ABB RobotStudio station: Assingmennt.rspag

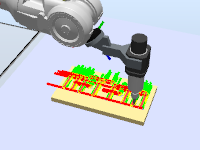
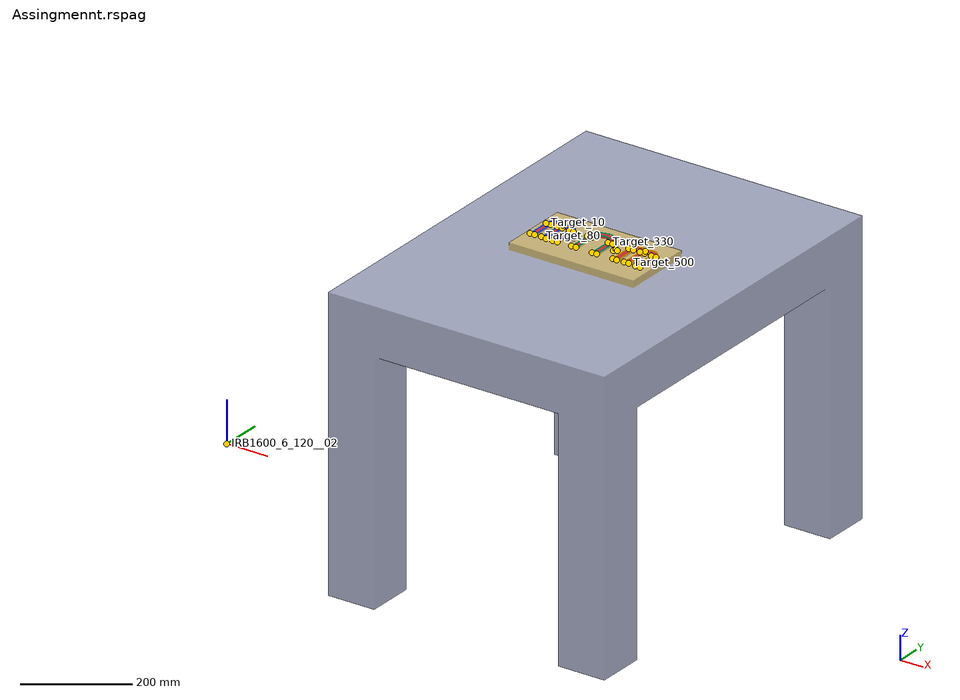
[picture v1: parts stored in the station drawn from their meshes, with robot base, taught points and paths (robot models come from the ABB library and are not in the file)]
--- station ---
Station Assingmennt (saved by RobotStudio 22.1.9826.0)
Controller IRB1600_6_120
  mechanical unit ROB_1: IRB1600_6_120__02, 6 joints, base frame (0, 0, 0) mm
Layout (positions relative to the parent item):
  - IRB1600_6_120__02 [mechanism, from Robots\IRB1600_6_120_G_02.rslib] at (0, 0, 0) mm; joint values [-0.0435, -0.0082, 0.1583, 0.0389, 0.7583, -0.0625] (rad or m)
  - MyTool [mechanism, from Training Objects\myTool.rslib] at (778.67, -32.12, 820.53) mm, rotated rx 180 ry 38 rz 180 deg
  - Table [part] at (800, 0, 0) mm, rotated rx 0 ry 0 rz 90 deg, size 800 x 600 x 600 mm
  - Part1 [part] at (800, 0, 600) mm, size 270 x 150 x 20 mm
Attachment: MyTool is attached to IRB1600_6_120__02 / Link6
Targets, tools, work objects and paths stored in the station and not in the controller backup, written as RAPID:
! task T_ROB1
MODULE Module1
  CONST robtarget Target_60:=[[202.210676312,424.371338975,20],[0,0,1,0],[0,0,0,0],[9E+09,9E+09,9E+09,9E+09,9E+09,9E+09]];
  CONST robtarget Target_120:=[[227.210676312,424.371338975,20],[0,0,1,0],[0,0,0,0],[9E+09,9E+09,9E+09,9E+09,9E+09,9E+09]];
  CONST robtarget Target_180:=[[222.399357136,434.659053801,20],[0,0,1,0],[0,0,0,0],[9E+09,9E+09,9E+09,9E+09,9E+09,9E+09]];
  CONST robtarget Target_210:=[[186.309791958,430.022914141,20],[0,0,1,0],[0,0,0,0],[9E+09,9E+09,9E+09,9E+09,9E+09,9E+09]];
  CONST robtarget Target_320:=[[307.210676312,433.031593012,20],[0,0,1,0],[0,0,0,0],[9E+09,9E+09,9E+09,9E+09,9E+09,9E+09]];
  CONST robtarget Target_380:=[[284.710676312,441.69184705,20],[0,0,1,0],[0,0,0,0],[9E+09,9E+09,9E+09,9E+09,9E+09,9E+09]];
  CONST robtarget Target_530:=[[406.25,424.371338975,20],[0,0,1,0],[0,0,0,0],[9E+09,9E+09,9E+09,9E+09,9E+09,9E+09]];
  CONST robtarget Target_590:=[[401.499668485,434.138320297,20],[0,0,1,0],[0,0,0,0],[9E+09,9E+09,9E+09,9E+09,9E+09,9E+09]];
  CONST robtarget Target_620:=[[365.571673376,430.19199697,20],[0,0,1,0],[0,0,0,0],[9E+09,9E+09,9E+09,9E+09,9E+09,9E+09]];
  CONST robtarget Target_680:=[[381.25,424.371338975,20],[0,0,1,0],[0,0,0,0],[9E+09,9E+09,9E+09,9E+09,9E+09,9E+09]];
ENDMODULE


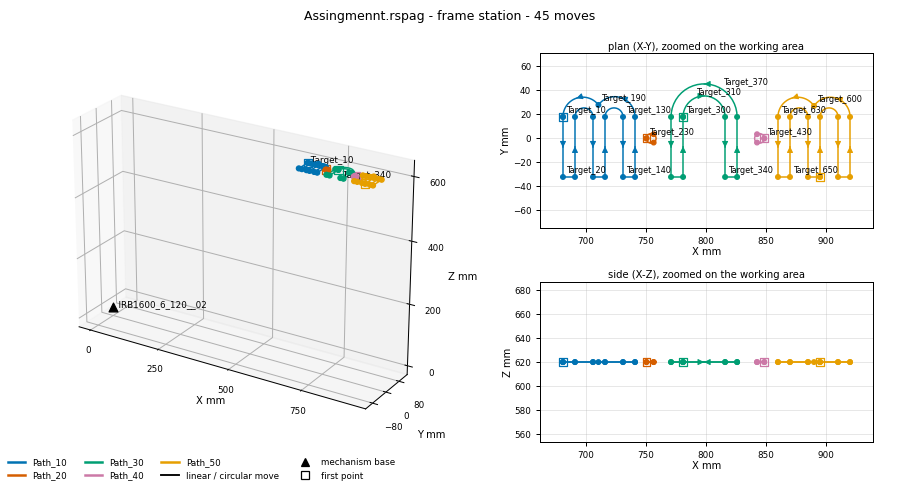
[picture p0: tool path of Assingmennt.rspag in frame station, 45 of 45 moves have a stored position in this frame; points joined in program order, loops and branches not executed]
--- Backups/IRB1600_6_120/RAPID/TASK1/PROGMOD/CalibData.mod ---
MODULE CalibData
    PERS tooldata MyTool:=[TRUE,[[31.792631019,0,229.638935148],[0.945518576,0,0.325568154,0]],[1,[0,0,1],[1,0,0,0],0,0,0]];
    PERS wobjdata Workobject_1:=[FALSE,TRUE,"",[[500,-400,600],[1,0,0,0]],[[0,0,0],[1,0,0,0]]];
ENDMODULE

--- Backups/IRB1600_6_120/RAPID/TASK1/PROGMOD/Module1.mod ---
MODULE Module1
    CONST robtarget Target_10:=[[180.960676312,417.876148446,20],[0,0,1,0],[0,0,0,0],[9E+09,9E+09,9E+09,9E+09,9E+09,9E+09]];
    CONST robtarget Target_20:=[[180.960676312,367.876148446,20],[0,0,1,0],[0,0,0,0],[9E+09,9E+09,9E+09,9E+09,9E+09,9E+09]];
    CONST robtarget Target_30:=[[190.960676312,367.876148446,20],[0,0,1,0],[0,0,0,0],[9E+09,9E+09,9E+09,9E+09,9E+09,9E+09]];
    CONST robtarget Target_40:=[[190.960676312,417.876148446,20],[0,0,1,0],[0,0,0,0],[9E+09,9E+09,9E+09,9E+09,9E+09,9E+09]];
    CONST robtarget Target_50:=[[194.710676312,424.371338975,20],[0,0,1,0],[0,0,0,0],[9E+09,9E+09,9E+09,9E+09,9E+09,9E+09]];
    CONST robtarget Target_70:=[[205.960676312,417.876148446,20],[0,0,1,0],[0,0,0,0],[9E+09,9E+09,9E+09,9E+09,9E+09,9E+09]];
    CONST robtarget Target_80:=[[205.960676312,367.876148446,20],[0,0,1,0],[0,0,0,0],[9E+09,9E+09,9E+09,9E+09,9E+09,9E+09]];
    CONST robtarget Target_90:=[[215.960676312,367.876148446,20],[0,0,1,0],[0,0,0,0],[9E+09,9E+09,9E+09,9E+09,9E+09,9E+09]];
    CONST robtarget Target_100:=[[215.960676312,417.876148446,20],[0,0,1,0],[0,0,0,0],[9E+09,9E+09,9E+09,9E+09,9E+09,9E+09]];
    CONST robtarget Target_110:=[[219.710676312,424.371338975,20],[0,0,1,0],[0,0,0,0],[9E+09,9E+09,9E+09,9E+09,9E+09,9E+09]];
    CONST robtarget Target_130:=[[230.960676312,417.876148446,20],[0,0,1,0],[0,0,0,0],[9E+09,9E+09,9E+09,9E+09,9E+09,9E+09]];
    CONST robtarget Target_140:=[[230.960676312,367.876148446,20],[0,0,1,0],[0,0,0,0],[9E+09,9E+09,9E+09,9E+09,9E+09,9E+09]];
    CONST robtarget Target_150:=[[240.960676312,367.876148446,20],[0,0,1,0],[0,0,0,0],[9E+09,9E+09,9E+09,9E+09,9E+09,9E+09]];
    CONST robtarget Target_160:=[[240.960676312,417.876148446,20],[0,0,1,0],[0,0,0,0],[9E+09,9E+09,9E+09,9E+09,9E+09,9E+09]];
    CONST robtarget Target_170:=[[235.405653207,430.388027618,20],[0,0,1,0],[0,0,0,0],[9E+09,9E+09,9E+09,9E+09,9E+09,9E+09]];
    CONST robtarget Target_190:=[[210.508284978,427.876148446,20],[0,0,1,0],[0,0,0,0],[9E+09,9E+09,9E+09,9E+09,9E+09,9E+09]];
    CONST robtarget Target_200:=[[198.881728,434.277720743,20],[0,0,1,0],[0,0,0,0],[9E+09,9E+09,9E+09,9E+09,9E+09,9E+09]];
    CONST robtarget Target_220:=[[180.960676312,417.876148446,20],[0,0,1,0],[0,0,0,0],[9E+09,9E+09,9E+09,9E+09,9E+09,9E+09]];
    CONST robtarget Target_230:=[[250.482336293,400,20],[0,0,1,0],[0,0,0,0],[9E+09,9E+09,9E+09,9E+09,9E+09,9E+09]];
    CONST robtarget Target_240:=[[252.482336293,403.464101615,20],[0,0,1,0],[0,0,0,0],[9E+09,9E+09,9E+09,9E+09,9E+09,9E+09]];
    CONST robtarget Target_250:=[[256.482336293,403.464101615,20],[0,0,1,0],[0,0,0,0],[9E+09,9E+09,9E+09,9E+09,9E+09,9E+09]];
    CONST robtarget Target_260:=[[258.482336293,400,20],[0,0,1,0],[0,0,0,0],[9E+09,9E+09,9E+09,9E+09,9E+09,9E+09]];
    CONST robtarget Target_270:=[[256.482336293,396.535898385,20],[0,0,1,0],[0,0,0,0],[9E+09,9E+09,9E+09,9E+09,9E+09,9E+09]];
    CONST robtarget Target_280:=[[252.482336293,396.535898385,20],[0,0,1,0],[0,0,0,0],[9E+09,9E+09,9E+09,9E+09,9E+09,9E+09]];
    CONST robtarget Target_290:=[[250.482336293,400,20],[0,0,1,0],[0,0,0,0],[9E+09,9E+09,9E+09,9E+09,9E+09,9E+09]];
    CONST robtarget Target_300:=[[280.960676312,417.876148446,20],[0,0,1,0],[0,0,0,0],[9E+09,9E+09,9E+09,9E+09,9E+09,9E+09]];
    CONST robtarget Target_310:=[[289.710676312,433.031593012,20],[0,0,1,0],[0,0,0,0],[9E+09,9E+09,9E+09,9E+09,9E+09,9E+09]];
    CONST robtarget Target_330:=[[315.960676312,417.876148446,20],[0,0,1,0],[0,0,0,0],[9E+09,9E+09,9E+09,9E+09,9E+09,9E+09]];
    CONST robtarget Target_340:=[[315.960676312,367.876148446,20],[0,0,1,0],[0,0,0,0],[9E+09,9E+09,9E+09,9E+09,9E+09,9E+09]];
    CONST robtarget Target_350:=[[325.960676312,367.876148446,20],[0,0,1,0],[0,0,0,0],[9E+09,9E+09,9E+09,9E+09,9E+09,9E+09]];
    CONST robtarget Target_360:=[[325.960676312,417.876148446,20],[0,0,1,0],[0,0,0,0],[9E+09,9E+09,9E+09,9E+09,9E+09,9E+09]];
    CONST robtarget Target_370:=[[312.210676312,441.69184705,20],[0,0,1,0],[0,0,0,0],[9E+09,9E+09,9E+09,9E+09,9E+09,9E+09]];
    CONST robtarget Target_390:=[[270.960676312,417.876148446,20],[0,0,1,0],[0,0,0,0],[9E+09,9E+09,9E+09,9E+09,9E+09,9E+09]];
    CONST robtarget Target_400:=[[270.960676312,367.876148446,20],[0,0,1,0],[0,0,0,0],[9E+09,9E+09,9E+09,9E+09,9E+09,9E+09]];
    CONST robtarget Target_410:=[[280.960676312,367.876148446,20],[0,0,1,0],[0,0,0,0],[9E+09,9E+09,9E+09,9E+09,9E+09,9E+09]];
    CONST robtarget Target_420:=[[280.960676312,417.876148446,20],[0,0,1,0],[0,0,0,0],[9E+09,9E+09,9E+09,9E+09,9E+09,9E+09]];
    CONST robtarget Target_430:=[[348.553180702,400,20],[0,0,1,0],[0,0,0,0],[9E+09,9E+09,9E+09,9E+09,9E+09,9E+09]];
    CONST robtarget Target_440:=[[346.553180702,396.535898385,20],[0,0,1,0],[0,0,0,0],[9E+09,9E+09,9E+09,9E+09,9E+09,9E+09]];
    CONST robtarget Target_450:=[[342.553180702,396.535898385,20],[0,0,1,0],[0,0,0,0],[9E+09,9E+09,9E+09,9E+09,9E+09,9E+09]];
    CONST robtarget Target_460:=[[340.553180702,400,20],[0,0,1,0],[0,0,0,0],[9E+09,9E+09,9E+09,9E+09,9E+09,9E+09]];
    CONST robtarget Target_470:=[[342.553180702,403.464101615,20],[0,0,1,0],[0,0,0,0],[9E+09,9E+09,9E+09,9E+09,9E+09,9E+09]];
    CONST robtarget Target_480:=[[346.553180702,403.464101615,20],[0,0,1,0],[0,0,0,0],[9E+09,9E+09,9E+09,9E+09,9E+09,9E+09]];
    CONST robtarget Target_490:=[[348.553180702,400,20],[0,0,1,0],[0,0,0,0],[9E+09,9E+09,9E+09,9E+09,9E+09,9E+09]];
    CONST robtarget Target_500:=[[395,367.876148446,20],[0,0,1,0],[0,0,0,0],[9E+09,9E+09,9E+09,9E+09,9E+09,9E+09]];
    CONST robtarget Target_510:=[[395,417.876148446,20],[0,0,1,0],[0,0,0,0],[9E+09,9E+09,9E+09,9E+09,9E+09,9E+09]];
    CONST robtarget Target_520:=[[398.75,424.371338975,20],[0,0,1,0],[0,0,0,0],[9E+09,9E+09,9E+09,9E+09,9E+09,9E+09]];
    CONST robtarget Target_540:=[[410,417.876148446,20],[0,0,1,0],[0,0,0,0],[9E+09,9E+09,9E+09,9E+09,9E+09,9E+09]];
    CONST robtarget Target_550:=[[410,367.876148446,20],[0,0,1,0],[0,0,0,0],[9E+09,9E+09,9E+09,9E+09,9E+09,9E+09]];
    CONST robtarget Target_560:=[[420,367.876148446,20],[0,0,1,0],[0,0,0,0],[9E+09,9E+09,9E+09,9E+09,9E+09,9E+09]];
    CONST robtarget Target_570:=[[420,417.876148446,20],[0,0,1,0],[0,0,0,0],[9E+09,9E+09,9E+09,9E+09,9E+09,9E+09]];
    CONST robtarget Target_580:=[[414.428326624,430.19199697,20],[0,0,1,0],[0,0,0,0],[9E+09,9E+09,9E+09,9E+09,9E+09,9E+09]];
    CONST robtarget Target_600:=[[390,427.03330138,20],[0,0,1,0],[0,0,0,0],[9E+09,9E+09,9E+09,9E+09,9E+09,9E+09]];
    CONST robtarget Target_610:=[[378.500331515,434.138320297,20],[0,0,1,0],[0,0,0,0],[9E+09,9E+09,9E+09,9E+09,9E+09,9E+09]];
    CONST robtarget Target_630:=[[360,417.876148446,20],[0,0,1,0],[0,0,0,0],[9E+09,9E+09,9E+09,9E+09,9E+09,9E+09]];
    CONST robtarget Target_640:=[[360,367.876148446,20],[0,0,1,0],[0,0,0,0],[9E+09,9E+09,9E+09,9E+09,9E+09,9E+09]];
    CONST robtarget Target_650:=[[370,367.876148446,20],[0,0,1,0],[0,0,0,0],[9E+09,9E+09,9E+09,9E+09,9E+09,9E+09]];
    CONST robtarget Target_660:=[[370,417.876148446,20],[0,0,1,0],[0,0,0,0],[9E+09,9E+09,9E+09,9E+09,9E+09,9E+09]];
    CONST robtarget Target_670:=[[373.75,424.371338975,20],[0,0,1,0],[0,0,0,0],[9E+09,9E+09,9E+09,9E+09,9E+09,9E+09]];
    CONST robtarget Target_690:=[[385,417.876148446,20],[0,0,1,0],[0,0,0,0],[9E+09,9E+09,9E+09,9E+09,9E+09,9E+09]];
    CONST robtarget Target_700:=[[385,367.876148446,20],[0,0,1,0],[0,0,0,0],[9E+09,9E+09,9E+09,9E+09,9E+09,9E+09]];
    CONST robtarget Target_710:=[[395,367.876148446,20],[0,0,1,0],[0,0,0,0],[9E+09,9E+09,9E+09,9E+09,9E+09,9E+09]];

    PROC main()
        Path_10;
        Path_20;
        Path_30;
        Path_40;
        Path_50;
    ENDPROC


    PROC Path_10()
        MoveL Target_10,v300,fine,MyTool\WObj:=Workobject_1;
        MoveL Target_20,v300,fine,MyTool\WObj:=Workobject_1;
        MoveL Target_30,v300,fine,MyTool\WObj:=Workobject_1;
        MoveL Target_40,v300,fine,MyTool\WObj:=Workobject_1;
        MoveC Target_50,Target_70,v300,fine,MyTool\WObj:=Workobject_1;
        MoveL Target_80,v300,fine,MyTool\WObj:=Workobject_1;
        MoveL Target_90,v300,fine,MyTool\WObj:=Workobject_1;
        MoveL Target_100,v300,fine,MyTool\WObj:=Workobject_1;
        MoveC Target_110,Target_130,v300,fine,MyTool\WObj:=Workobject_1;
        MoveL Target_140,v300,fine,MyTool\WObj:=Workobject_1;
        MoveL Target_150,v300,fine,MyTool\WObj:=Workobject_1;
        MoveL Target_160,v300,fine,MyTool\WObj:=Workobject_1;
        MoveC Target_170,Target_190,v300,fine,MyTool\WObj:=Workobject_1;
        MoveC Target_200,Target_220,v300,fine,MyTool\WObj:=Workobject_1;
    ENDPROC
    PROC Path_20()
        MoveL Target_230,v40,fine,MyTool\WObj:=Workobject_1;
        MoveC Target_240,Target_250,v40,fine,MyTool\WObj:=Workobject_1;
        MoveC Target_260,Target_270,v40,fine,MyTool\WObj:=Workobject_1;
        MoveC Target_280,Target_290,v40,fine,MyTool\WObj:=Workobject_1;
    ENDPROC
    PROC Path_30()
        MoveL Target_300,v100,fine,MyTool\WObj:=Workobject_1;
        MoveC Target_310,Target_330,v100,fine,MyTool\WObj:=Workobject_1;
        MoveL Target_340,v100,fine,MyTool\WObj:=Workobject_1;
        MoveL Target_350,v100,fine,MyTool\WObj:=Workobject_1;
        MoveL Target_360,v100,fine,MyTool\WObj:=Workobject_1;
        MoveC Target_370,Target_390,v100,fine,MyTool\WObj:=Workobject_1;
        MoveL Target_400,v100,fine,MyTool\WObj:=Workobject_1;
        MoveL Target_410,v100,fine,MyTool\WObj:=Workobject_1;
        MoveL Target_420,v100,fine,MyTool\WObj:=Workobject_1;
    ENDPROC
    PROC Path_40()
        MoveL Target_430,v50,fine,MyTool\WObj:=Workobject_1;
        MoveC Target_440,Target_450,v50,fine,MyTool\WObj:=Workobject_1;
        MoveC Target_460,Target_470,v50,fine,MyTool\WObj:=Workobject_1;
        MoveC Target_480,Target_490,v50,fine,MyTool\WObj:=Workobject_1;
    ENDPROC
    PROC Path_50()
        MoveL Target_500,v100,fine,MyTool\WObj:=Workobject_1;
        MoveL Target_510,v100,fine,MyTool\WObj:=Workobject_1;
        MoveC Target_520,Target_540,v100,fine,MyTool\WObj:=Workobject_1;
        MoveL Target_550,v100,fine,MyTool\WObj:=Workobject_1;
        MoveL Target_560,v100,fine,MyTool\WObj:=Workobject_1;
        MoveL Target_570,v100,fine,MyTool\WObj:=Workobject_1;
        MoveC Target_580,Target_600,v100,fine,MyTool\WObj:=Workobject_1;
        MoveC Target_610,Target_630,v100,fine,MyTool\WObj:=Workobject_1;
        MoveL Target_640,v100,fine,MyTool\WObj:=Workobject_1;
        MoveL Target_650,v100,fine,MyTool\WObj:=Workobject_1;
        MoveL Target_660,v100,fine,MyTool\WObj:=Workobject_1;
        MoveC Target_670,Target_690,v100,fine,MyTool\WObj:=Workobject_1;
        MoveL Target_700,v100,fine,MyTool\WObj:=Workobject_1;
        MoveL Target_710,v100,fine,MyTool\WObj:=Workobject_1;
    ENDPROC
ENDMODULE
